Omron CX-Programmer project 新工程 (CX-Programmer 9.73)

# PLC InjectionMoldingmachine_CY200: CPM1(CPM1A) CPU40

## Global symbols (name address type ; comment)
0.01 BOOL  ; 调模PB
0.02 BOOL  ; 开始PB
0.03 BOOL  ; 电眼PH
0.04 BOOL  ; 射出PB
0.06 BOOL  ; 顶退PB
0.07 BOOL  ; 顶出
0.08 BOOL  ; 加料PB
0.11 BOOL  ; 自动选用SW
10.00 BOOL  ; 关慢阀
10.01 BOOL  ; 冷却计时器
10.02 BOOL  ; 关快阀
10.03 BOOL  ; 低压阀
10.04 BOOL  ; 顶出阀
10.05 BOOL  ; 加料阀
10.06 BOOL  ; 顶退阀
10.07 BOOL  ; 松退阀（松退计时器）
11.00 BOOL  ; 开模阀
11.01 BOOL  ; 关模阀
11.02 BOOL  ; 总压阀
11.03 BOOL  ; 引阀
11.04 BOOL  ; 一压阀
11.05 BOOL  ; 二压阀
11.06 BOOL  ; 射出阀
11.07 BOOL  ; 温度报警
1.00 BOOL  ; 关慢PS
1.01 BOOL  ; 急停PB
1.02 BOOL  ; 开止PS
1.03 BOOL  ; 冷料
1.04 BOOL  ; 关高压PS
1.05 BOOL  ; 松退PB
1.06 BOOL  ; 射二压PS
1.07 BOOL  ; 顶出PB
1.08 BOOL  ; 加料止PS
1.09 BOOL  ; 松退止PS
1.10 BOOL  ; 冷却计时到
1.11 BOOL  ; 射出计时到

## Program 新程序1 (no task)
; 概况： / 这个PLC程序实现了一个15T立式注塑机的控制系统，应用于塑料制品生产车间，用于控制注塑机的模具开合、射出、顶出、冷却等动作，确保塑料制品的自动化成型。 / 系统包含故障检测功能，如温度报警监测温度异常，急停按钮用于紧急停止所有动作。 / 系统包含操作面板按钮，如开始按钮、调模按钮、射出按钮、顶出按钮、加料按钮和急停按钮。 / 系统还包括传感器，如电眼传感器、开止传感器、关慢传感器、关高压传感器和加料止传感器，以及执行器，如关模阀、开模阀、射出阀、顶出阀和加料阀。 / 系统的目标效果： / 在自动模式下，通过自动模式开关启用后，按下开始按钮，系统在关模启动前检查电眼传感器，若无障碍物则激活关模阀。关模过程中依赖初始检查确保安全。关模进入慢速阶段时，关慢传感器置位，激活关慢阀；进入高压阶段时，关高压传感器置位，激活低压阀，确保关模平稳安全。系统设计避免关模阀和开模阀同时激活，以防止模具动作冲突。 / 关模完成后，系统执行射出动作，激活射出阀，将熔融塑料注入模具。射出可由射出按钮手动触发或自动流程控制，射二压传感器置位时激活二压阀，射出计时到时结束。若温度报警置位，系统将继续射出动作，需注意温度异常可能影响产品质量。当系统运行时间过长，温度报警会提示操作员检查设备状态。 / 射出结束后，冷却计时器启动，进入冷却阶段。冷却计时到未置位前，系统仍可激活开模阀，需确保塑料充分冷却以避免变形。冷却计时到置位后，系统确认冷却阶段结束，准备后续动作。冷却完成后，系统打开开模阀，开止传感器置位时停止开模。模具打开后，顶出阀激活。顶出动作可由顶出按钮1手动触发，完成后通过顶退按钮激活顶退阀回退顶针。 / 加料动作由加料按钮触发，激活加料阀，加料止传感器置位时停止，确保料斗适量填充塑料颗粒。松退按钮可触发松退阀，辅助模具松开。 / 任何时候，按下急停按钮，系统将重置流程，但输出阀门可能不会立即关闭，需注意紧急情况下的安全。

### Section 段1

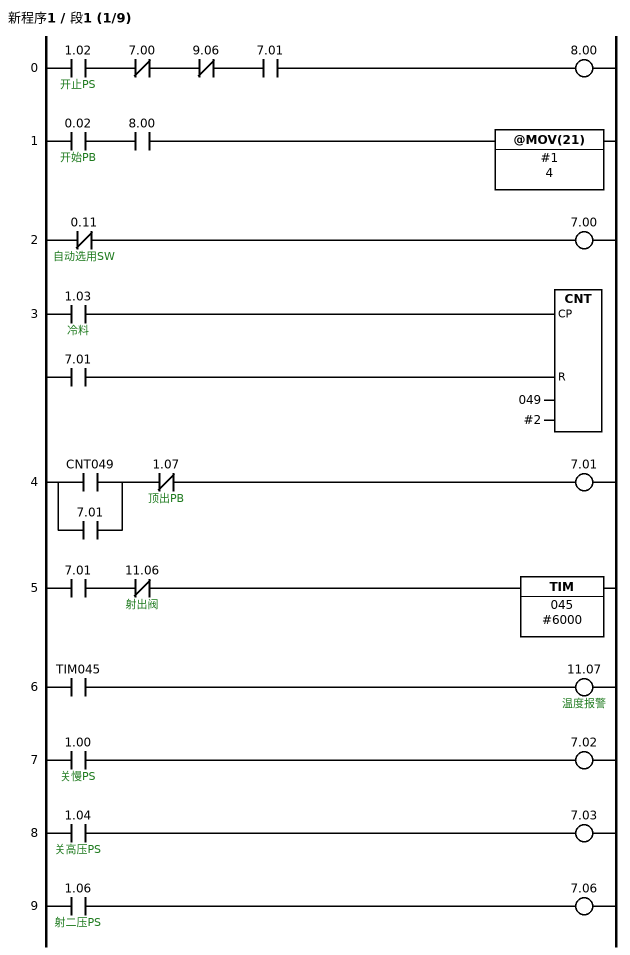
; rung 0
LD 1.02  ; 开止PS
ANDNOT 7.00
ANDNOT 9.06
AND 7.01
OUT 8.00
; rung 1
LD 0.02  ; 开始PB
AND 8.00
@MOV(21) #1 4
; rung 2
LDNOT 0.11  ; 自动选用SW
OUT 7.00
; rung 3
LD 1.03  ; 冷料
LD 7.01
CNT 049 #2
; rung 4
LD CNT049
OR 7.01
ANDNOT 1.07  ; 顶出PB
OUT 7.01
; rung 5
LD 7.01
ANDNOT 11.06  ; 射出阀
TIM 045 #6000
; rung 6
LD TIM045
OUT 11.07  ; 温度报警
; rung 7
LD 1.00  ; 关慢PS
OUT 7.02
; rung 8
LD 1.04  ; 关高压PS
OUT 7.03
; rung 9
LD 1.06  ; 射二压PS
OUT 7.06

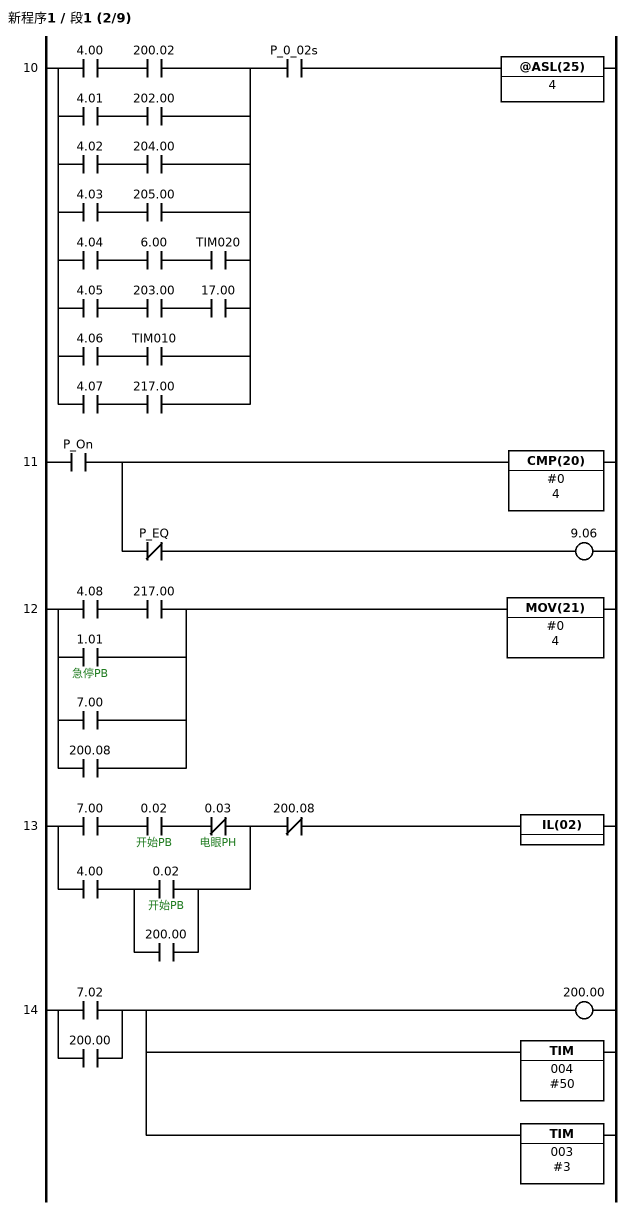
; rung 10
LD 4.00
AND 200.02
LD 4.01
AND 202.00
ORLD
LD 4.02
AND 204.00
ORLD
LD 4.03
AND 205.00
ORLD
LD 4.04
AND 6.00
AND TIM020
ORLD
LD 4.05
AND 203.00
AND 17.00
ORLD
LD 4.06
AND TIM010
ORLD
LD 4.07
AND 217.00
ORLD
AND P_0_02s
@ASL(25) 4
; rung 11
LD P_On
CMP(20) #0 4
ANDNOT P_EQ
OUT 9.06
; rung 12
LD 4.08
AND 217.00
OR 1.01  ; 急停PB
OR 7.00
OR 200.08
MOV(21) #0 4
; rung 13
LD 7.00
AND 0.02  ; 开始PB
ANDNOT 0.03  ; 电眼PH
LD 4.00
LD 0.02  ; 开始PB
OR 200.00
ANDLD
ORLD
ANDNOT 200.08
IL(02)
; rung 14
LD 7.02
OR 200.00
OUT 200.00
TIM 004 #50
TIM 003 #3

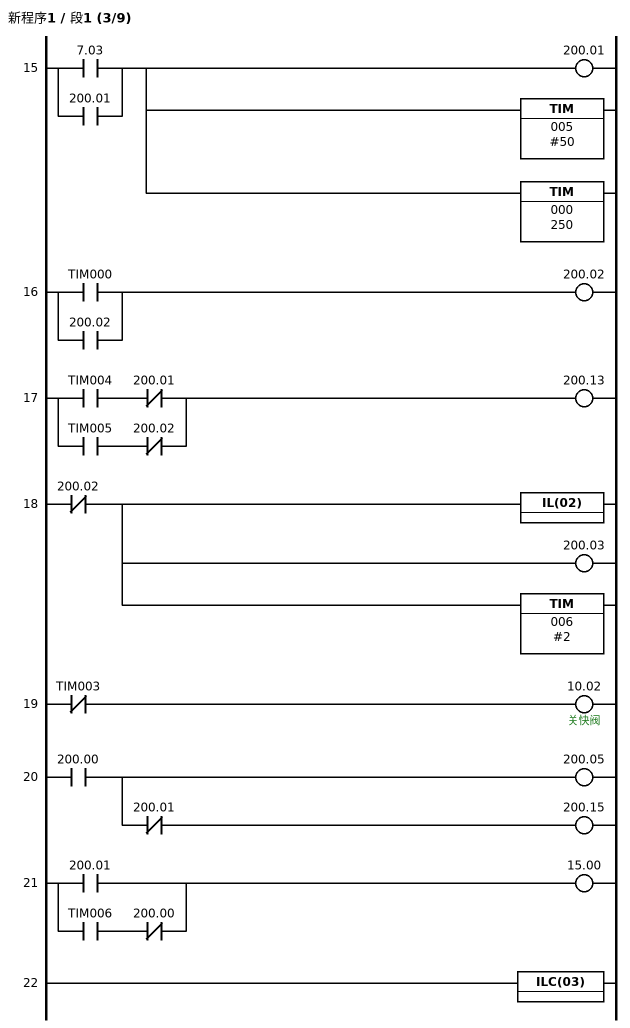
; rung 15
LD 7.03
OR 200.01
OUT 200.01
TIM 005 #50
TIM 000 250
; rung 16
LD TIM000
OR 200.02
OUT 200.02
; rung 17
LD TIM004
ANDNOT 200.01
LD TIM005
ANDNOT 200.02
ORLD
OUT 200.13
; rung 18
LDNOT 200.02
IL(02)
OUT 200.03
TIM 006 #2
; rung 19
LDNOT TIM003
OUT 10.02  ; 关快阀
; rung 20
LD 200.00
OUT 200.05
ANDNOT 200.01
OUT 200.15
; rung 21
LD 200.01
LD TIM006
ANDNOT 200.00
ORLD
OUT 15.00
; rung 22
ILC(03)

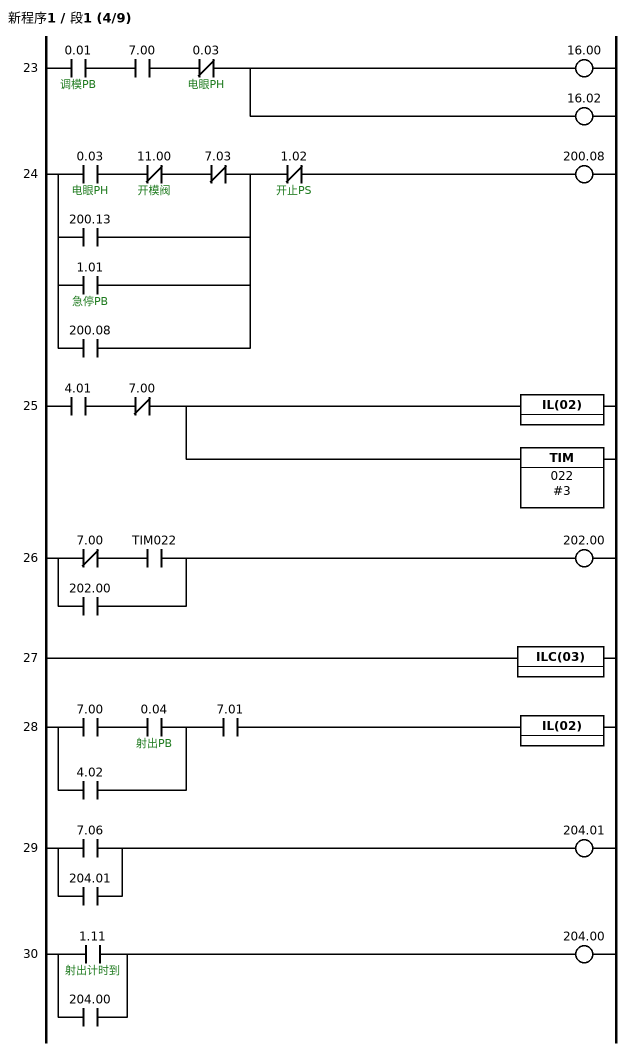
; rung 23
LD 0.01  ; 调模PB
AND 7.00
ANDNOT 0.03  ; 电眼PH
OUT 16.00
OUT 16.02
; rung 24
LD 0.03  ; 电眼PH
ANDNOT 11.00  ; 开模阀
ANDNOT 7.03
OR 200.13
OR 1.01  ; 急停PB
OR 200.08
ANDNOT 1.02  ; 开止PS
OUT 200.08
; rung 25
LD 4.01
ANDNOT 7.00
IL(02)
TIM 022 #3
; rung 26
LDNOT 7.00
AND TIM022
OR 202.00
OUT 202.00
; rung 27
ILC(03)
; rung 28
LD 7.00
AND 0.04  ; 射出PB
OR 4.02
AND 7.01
IL(02)
; rung 29
LD 7.06
OR 204.01
OUT 204.01
; rung 30
LD 1.11  ; 射出计时到
OR 204.00
OUT 204.00

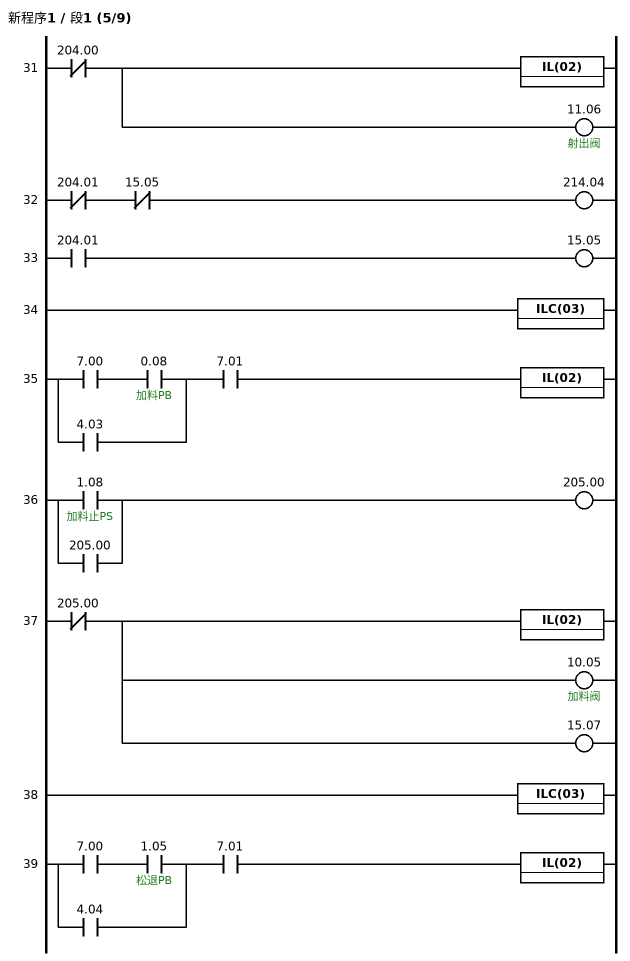
; rung 31
LDNOT 204.00
IL(02)
OUT 11.06  ; 射出阀
; rung 32
LDNOT 204.01
ANDNOT 15.05
OUT 214.04
; rung 33
LD 204.01
OUT 15.05
; rung 34
ILC(03)
; rung 35
LD 7.00
AND 0.08  ; 加料PB
OR 4.03
AND 7.01
IL(02)
; rung 36
LD 1.08  ; 加料止PS
OR 205.00
OUT 205.00
; rung 37
LDNOT 205.00
IL(02)
OUT 10.05  ; 加料阀
OUT 15.07
; rung 38
ILC(03)
; rung 39
LD 7.00
AND 1.05  ; 松退PB
OR 4.04
AND 7.01
IL(02)

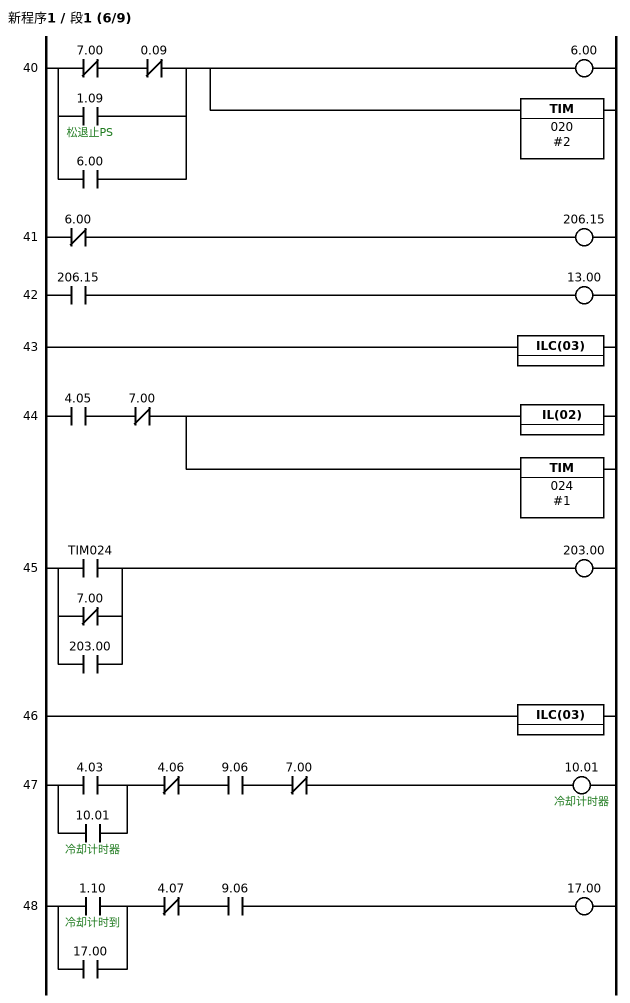
; rung 40
LDNOT 7.00
ANDNOT 0.09
OR 1.09  ; 松退止PS
OR 6.00
OUT 6.00
TIM 020 #2
; rung 41
LDNOT 6.00
OUT 206.15
; rung 42
LD 206.15
OUT 13.00
; rung 43
ILC(03)
; rung 44
LD 4.05
ANDNOT 7.00
IL(02)
TIM 024 #1
; rung 45
LD TIM024
ORNOT 7.00
OR 203.00
OUT 203.00
; rung 46
ILC(03)
; rung 47
LD 4.03
OR 10.01  ; 冷却计时器
ANDNOT 4.06
AND 9.06
ANDNOT 7.00
OUT 10.01  ; 冷却计时器
; rung 48
LD 1.10  ; 冷却计时到
OR 17.00
ANDNOT 4.07
AND 9.06
OUT 17.00

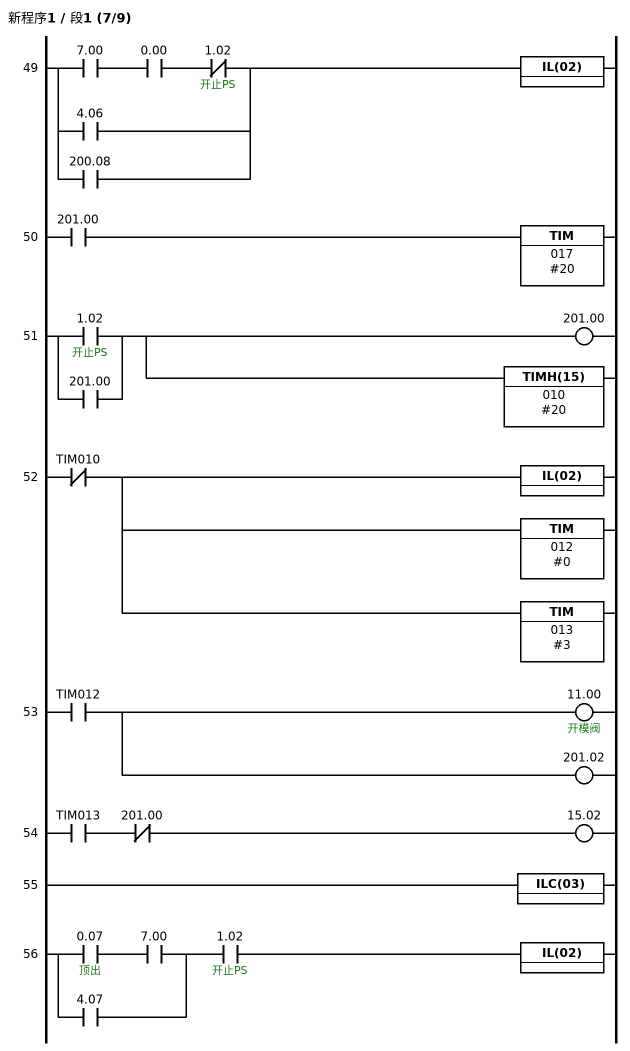
; rung 49
LD 7.00
AND 0.00
ANDNOT 1.02  ; 开止PS
OR 4.06
OR 200.08
IL(02)
; rung 50
LD 201.00
TIM 017 #20
; rung 51
LD 1.02  ; 开止PS
OR 201.00
OUT 201.00
TIMH(15) 010 #20
; rung 52
LDNOT TIM010
IL(02)
TIM 012 #0
TIM 013 #3
; rung 53
LD TIM012
OUT 11.00  ; 开模阀
OUT 201.02
; rung 54
LD TIM013
ANDNOT 201.00
OUT 15.02
; rung 55
ILC(03)
; rung 56
LD 0.07  ; 顶出
AND 7.00
OR 4.07
AND 1.02  ; 开止PS
IL(02)

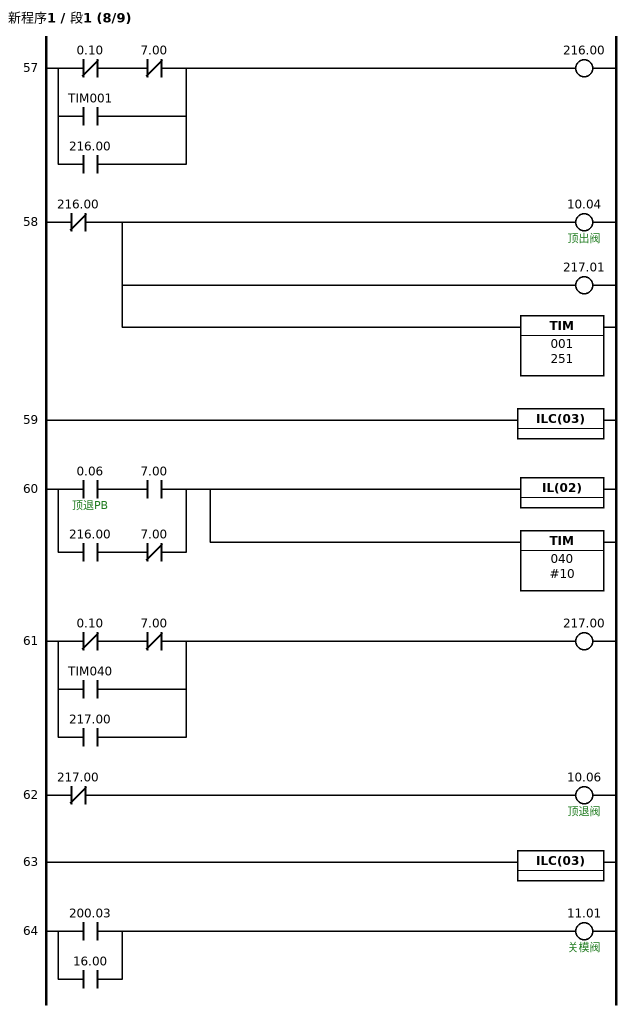
; rung 57
LDNOT 0.10
ANDNOT 7.00
OR TIM001
OR 216.00
OUT 216.00
; rung 58
LDNOT 216.00
OUT 10.04  ; 顶出阀
OUT 217.01
TIM 001 251
; rung 59
ILC(03)
; rung 60
LD 0.06  ; 顶退PB
AND 7.00
LD 216.00
ANDNOT 7.00
ORLD
IL(02)
TIM 040 #10
; rung 61
LDNOT 0.10
ANDNOT 7.00
OR TIM040
OR 217.00
OUT 217.00
; rung 62
LDNOT 217.00
OUT 10.06  ; 顶退阀
; rung 63
ILC(03)
; rung 64
LD 200.03
OR 16.00
OUT 11.01  ; 关模阀

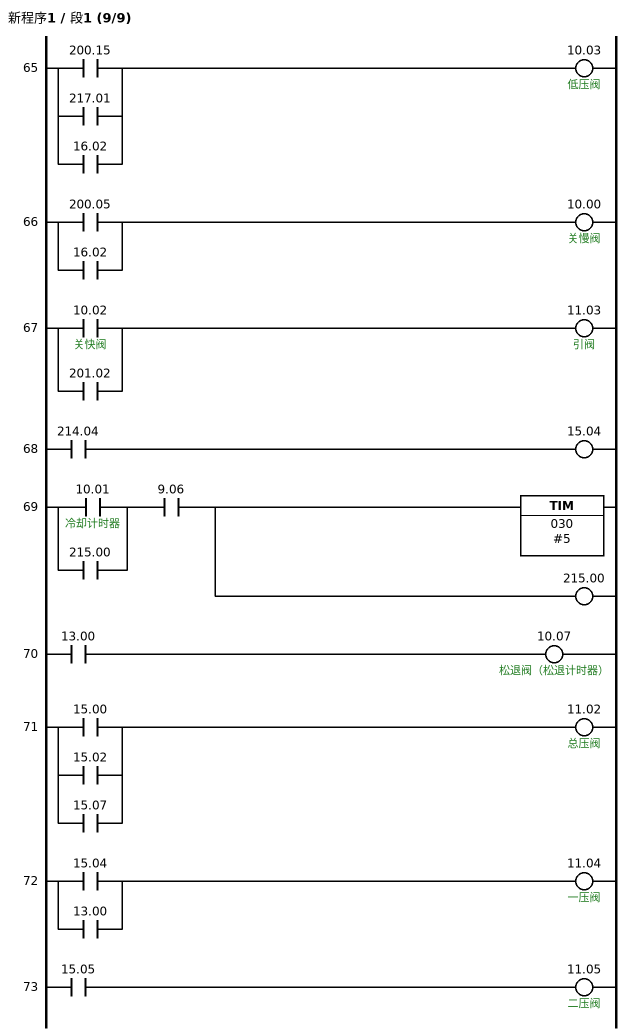
; rung 65
LD 200.15
OR 217.01
OR 16.02
OUT 10.03  ; 低压阀
; rung 66
LD 200.05
OR 16.02
OUT 10.00  ; 关慢阀
; rung 67
LD 10.02  ; 关快阀
OR 201.02
OUT 11.03  ; 引阀
; rung 68
LD 214.04
OUT 15.04
; rung 69
LD 10.01  ; 冷却计时器
OR 215.00
AND 9.06
TIM 030 #5
OUT 215.00
; rung 70
LD 13.00
OUT 10.07  ; 松退阀（松退计时器）
; rung 71
LD 15.00
OR 15.02
OR 15.07
OUT 11.02  ; 总压阀
; rung 72
LD 15.04
OR 13.00
OUT 11.04  ; 一压阀
; rung 73
LD 15.05
OUT 11.05  ; 二压阀
; rung 74
END(01)